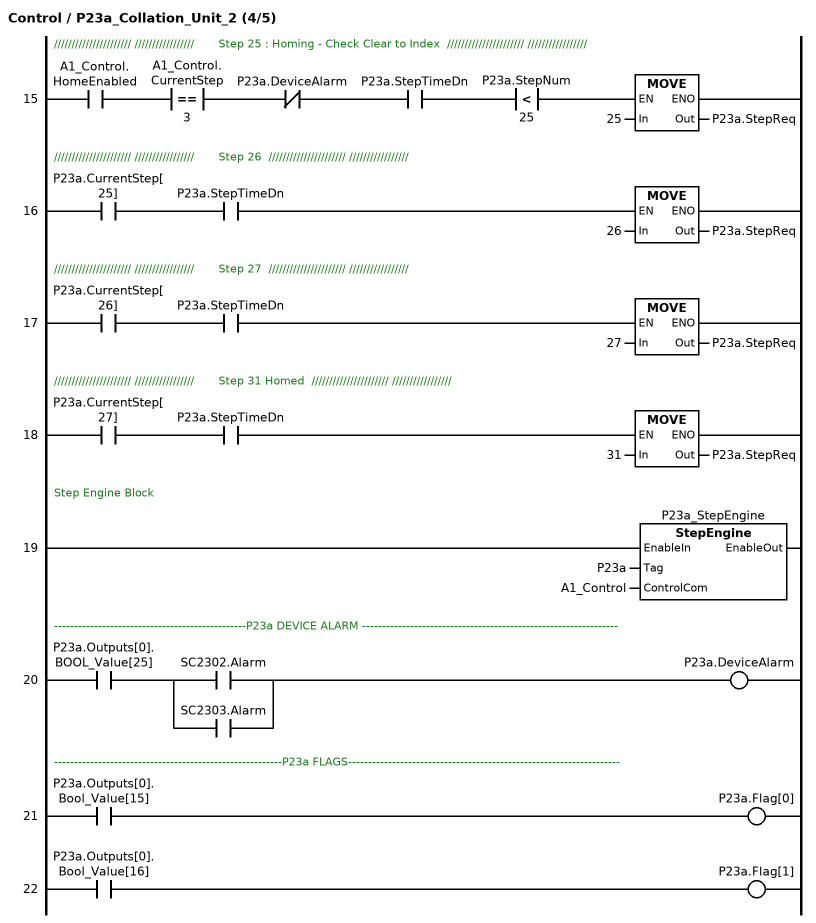
(* [picture p48: Control / P23a_Collation_Unit_2, rungs 15-22] *)
(* Rung 15: ////////////////////// /////////////////       Step 25 : Homing - Check Clear to Index  ////////////////////// ///////////////// *)
IF A1_Control.HomeEnabled AND (A1_Control.CurrentStep = 3) AND NOT P23a.DeviceAlarm AND P23a.StepTimeDn AND (P23a.StepNum < 25) THEN
    P23a.StepReq := 25;
END_IF;
(* Rung 16: ////////////////////// /////////////////       Step 26  ////////////////////// ///////////////// *)
IF P23a.CurrentStep[25] AND P23a.StepTimeDn THEN P23a.StepReq := 26; END_IF;
(* Rung 17: ////////////////////// /////////////////       Step 27  ////////////////////// ///////////////// *)
IF P23a.CurrentStep[26] AND P23a.StepTimeDn THEN P23a.StepReq := 27; END_IF;
(* Rung 18: ////////////////////// /////////////////       Step 31 Homed  ////////////////////// ///////////////// *)
IF P23a.CurrentStep[27] AND P23a.StepTimeDn THEN P23a.StepReq := 31; END_IF;
(* Rung 19: Step Engine Block *)
P23a_StepEngine(EnableIn := TRUE, Tag := P23a, ControlCom := A1_Control);
(* Rung 20: ------------------------------------------------P23a DEVICE ALARM ---------------------------------------------------------------- *)
P23a.DeviceAlarm := P23a.Outputs[0].BOOL_Value[25] AND (SC2302.Alarm OR SC2303.Alarm);
(* Rung 21: ---------------------------------------------------------P23a FLAGS-------------------------------------------------------------------- *)
P23a.Flag[0] := P23a.Outputs[0].Bool_Value[15];
(* Rung 22 *)
P23a.Flag[1] := P23a.Outputs[0].Bool_Value[16];

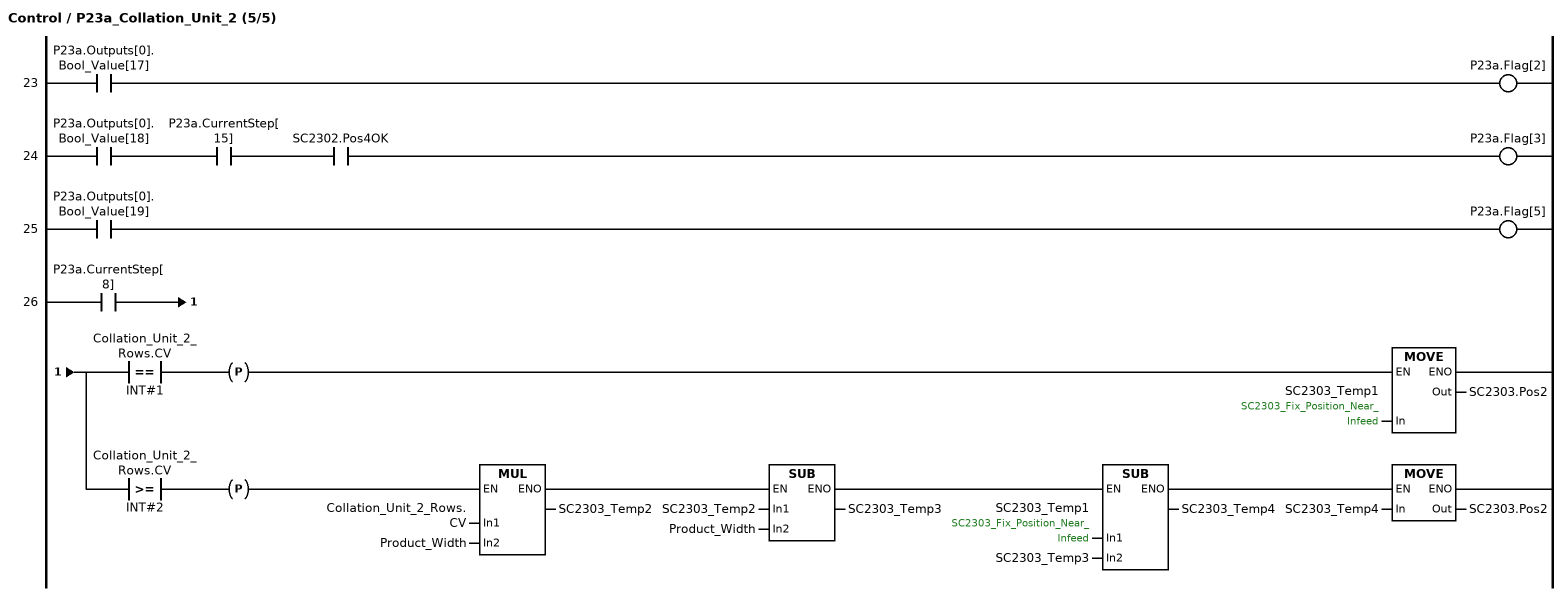
(* Rung 23 *)
P23a.Flag[2] := P23a.Outputs[0].Bool_Value[17];
(* Rung 24 *)
P23a.Flag[3] := P23a.Outputs[0].Bool_Value[18] AND P23a.CurrentStep[15] AND SC2302.Pos4OK;
(* notes on elements: Flag to Infeed conveyor *)
(* Rung 25 *)
P23a.Flag[5] := P23a.Outputs[0].Bool_Value[19];
(* Rung 26 *)
_e52(CLK := P23a.CurrentStep[8] AND (Collation_Unit_2_Rows.CV = INT#1));
IF _e52.Q THEN SC2303.Pos2 := SC2303_Temp1; END_IF;
_e53(CLK := P23a.CurrentStep[8] AND (Collation_Unit_2_Rows.CV >= INT#2));
IF _e53.Q THEN
    SC2303_Temp2 := Collation_Unit_2_Rows.CV * Product_Width;
    SC2303_Temp3 := SC2303_Temp2 - Product_Width;
    SC2303_Temp4 := SC2303_Temp1 - SC2303_Temp3;
    SC2303.Pos2 := SC2303_Temp4;
END_IF;

(* Section P17_MainDrive: ladder, written here as Structured Text *)

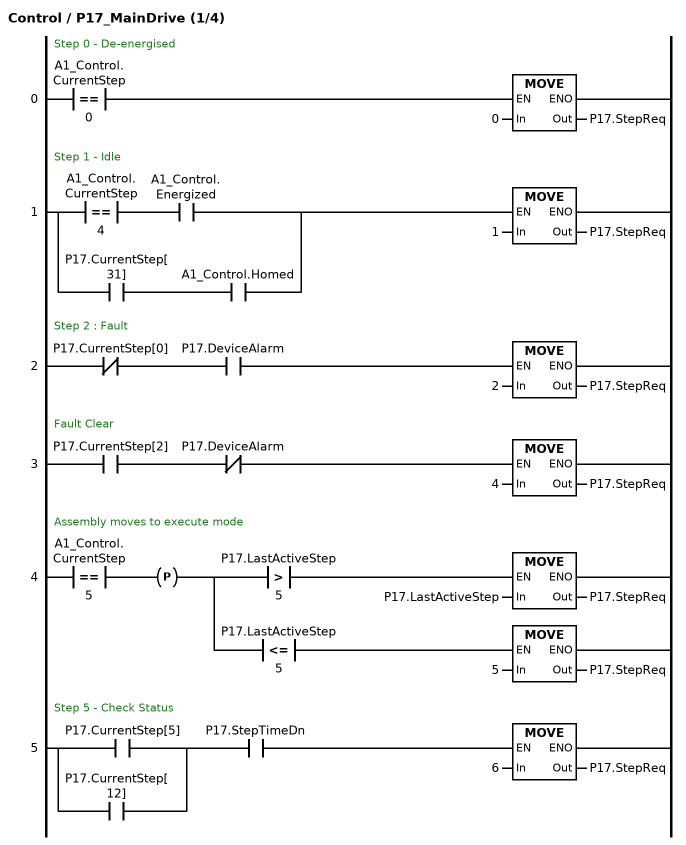
(* Rung 0: Step 0 - De-energised *)
IF A1_Control.CurrentStep = 0 THEN P17.StepReq := 0; END_IF;
(* Rung 1: Step 1 - Idle *)
IF ((A1_Control.CurrentStep = 4) AND A1_Control.Energized) OR (P17.CurrentStep[31] AND A1_Control.Homed) THEN
    P17.StepReq := 1;
END_IF;
(* Rung 2: Step 2 : Fault *)
IF NOT P17.CurrentStep[0] AND P17.DeviceAlarm THEN P17.StepReq := 2; END_IF;
(* Rung 3: Fault Clear *)
IF P17.CurrentStep[2] AND NOT P17.DeviceAlarm THEN P17.StepReq := 4; END_IF;
(* Rung 4: Assembly moves to execute mode *)
_e54(CLK := A1_Control.CurrentStep = 5);
IF _e54.Q AND (P17.LastActiveStep > 5) THEN P17.StepReq := P17.LastActiveStep; END_IF;
IF _e54.Q AND (P17.LastActiveStep <= 5) THEN P17.StepReq := 5; END_IF;
(* Rung 5: Step 5 - Check Status *)
IF (P17.CurrentStep[5] OR P17.CurrentStep[12]) AND P17.StepTimeDn THEN P17.StepReq := 6; END_IF;

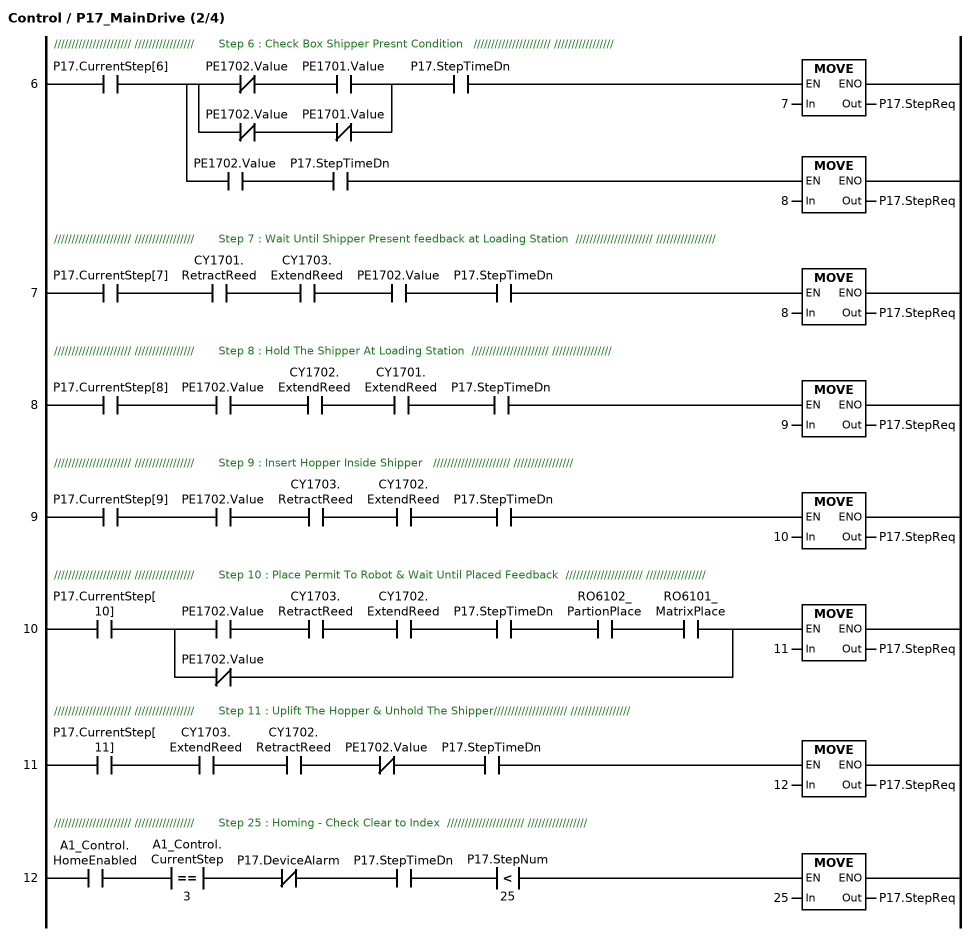
(* Rung 6: ////////////////////// /////////////////       Step 6 : Check Box Shipper Presnt Condition   ////////////////////// ///////////////// *)
_p55 := P17.CurrentStep[6];
IF P17.CurrentStep[6] AND ((NOT PE1702.Value AND PE1701.Value) OR (NOT PE1702.Value AND NOT PE1701.Value)) AND P17.StepTimeDn THEN
    P17.StepReq := 7;
END_IF;
IF _p55 AND PE1702.Value AND P17.StepTimeDn THEN P17.StepReq := 8; END_IF;
(* Rung 7: ////////////////////// /////////////////       Step 7 : Wait Until Shipper Present feedback at Loading Station  ////////////////////// ///////////////// *)
IF P17.CurrentStep[7] AND CY1701.RetractReed AND CY1703.ExtendReed AND PE1702.Value AND P17.StepTimeDn THEN
    P17.StepReq := 8;
END_IF;
(* Rung 8: ////////////////////// /////////////////       Step 8 : Hold The Shipper At Loading Station  ////////////////////// ///////////////// *)
IF P17.CurrentStep[8] AND PE1702.Value AND CY1702.ExtendReed AND CY1701.ExtendReed AND P17.StepTimeDn THEN
    P17.StepReq := 9;
END_IF;
(* Rung 9: ////////////////////// /////////////////       Step 9 : Insert Hopper Inside Shipper   ////////////////////// ///////////////// *)
IF P17.CurrentStep[9] AND PE1702.Value AND CY1703.RetractReed AND CY1702.ExtendReed AND P17.StepTimeDn THEN
    P17.StepReq := 10;
END_IF;
(* Rung 10: ////////////////////// /////////////////       Step 10 : Place Permit To Robot & Wait Until Placed Feedback  ////////////////////// ///////////////// *)
IF P17.CurrentStep[10] AND ((PE1702.Value AND CY1703.RetractReed AND CY1702.ExtendReed AND P17.StepTimeDn AND RO6102_PartionPlace AND RO6101_MatrixPlace) OR NOT PE1702.Value) THEN
    P17.StepReq := 11;
END_IF;
(* Rung 11: ////////////////////// /////////////////       Step 11 : Uplift The Hopper & Unhold The Shipper///////////////////// ///////////////// *)
IF P17.CurrentStep[11] AND CY1703.ExtendReed AND CY1702.RetractReed AND NOT PE1702.Value AND P17.StepTimeDn THEN
    P17.StepReq := 12;
END_IF;
(* Rung 12: ////////////////////// /////////////////       Step 25 : Homing - Check Clear to Index  ////////////////////// ///////////////// *)
IF A1_Control.HomeEnabled AND (A1_Control.CurrentStep = 3) AND NOT P17.DeviceAlarm AND P17.StepTimeDn AND (P17.StepNum < 25) THEN
    P17.StepReq := 25;
END_IF;

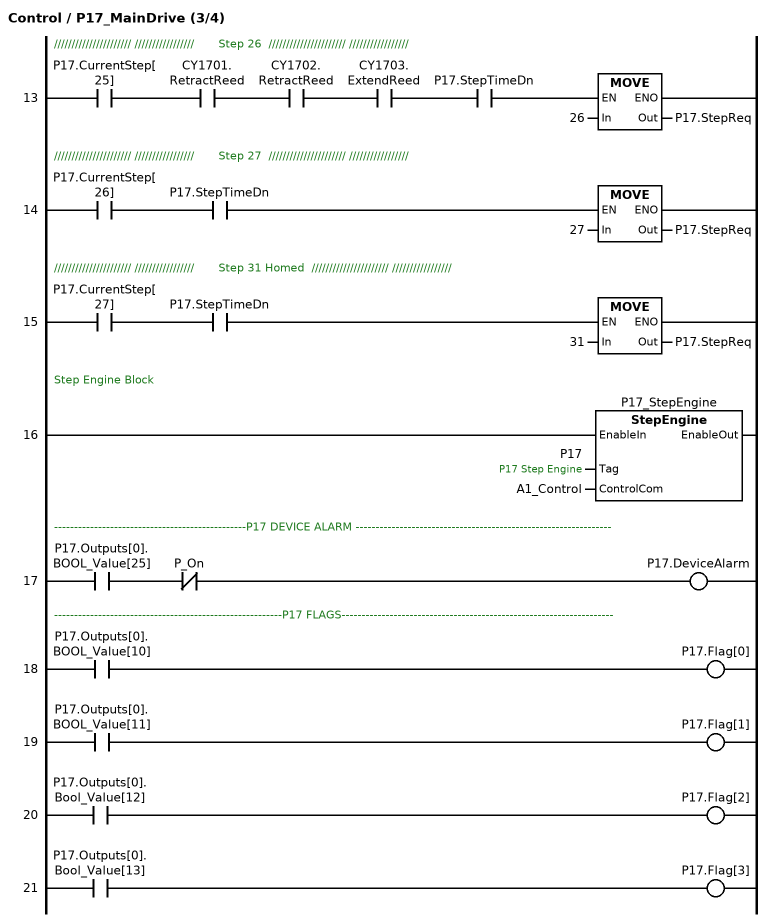
(* Rung 13: ////////////////////// /////////////////       Step 26  ////////////////////// ///////////////// *)
IF P17.CurrentStep[25] AND CY1701.RetractReed AND CY1702.RetractReed AND CY1703.ExtendReed AND P17.StepTimeDn THEN
    P17.StepReq := 26;
END_IF;
(* Rung 14: ////////////////////// /////////////////       Step 27  ////////////////////// ///////////////// *)
IF P17.CurrentStep[26] AND P17.StepTimeDn THEN P17.StepReq := 27; END_IF;
(* Rung 15: ////////////////////// /////////////////       Step 31 Homed  ////////////////////// ///////////////// *)
IF P17.CurrentStep[27] AND P17.StepTimeDn THEN P17.StepReq := 31; END_IF;
(* Rung 16: Step Engine Block *)
P17_StepEngine(EnableIn := TRUE, Tag := P17, ControlCom := A1_Control);
(* Rung 17: ------------------------------------------------P17 DEVICE ALARM ---------------------------------------------------------------- *)
P17.DeviceAlarm := P17.Outputs[0].BOOL_Value[25] AND NOT P_On;
(* Rung 18: ---------------------------------------------------------P17 FLAGS-------------------------------------------------------------------- *)
P17.Flag[0] := P17.Outputs[0].BOOL_Value[10];
(* Rung 19 *)
P17.Flag[1] := P17.Outputs[0].BOOL_Value[11];
(* Rung 20 *)
P17.Flag[2] := P17.Outputs[0].Bool_Value[12];
(* Rung 21 *)
P17.Flag[3] := P17.Outputs[0].Bool_Value[13];

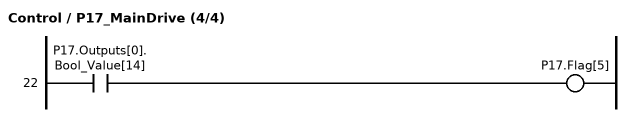
(* Rung 22 *)
P17.Flag[5] := P17.Outputs[0].Bool_Value[14];

(* Section P27_TopTapping: ladder, written here as Structured Text *)

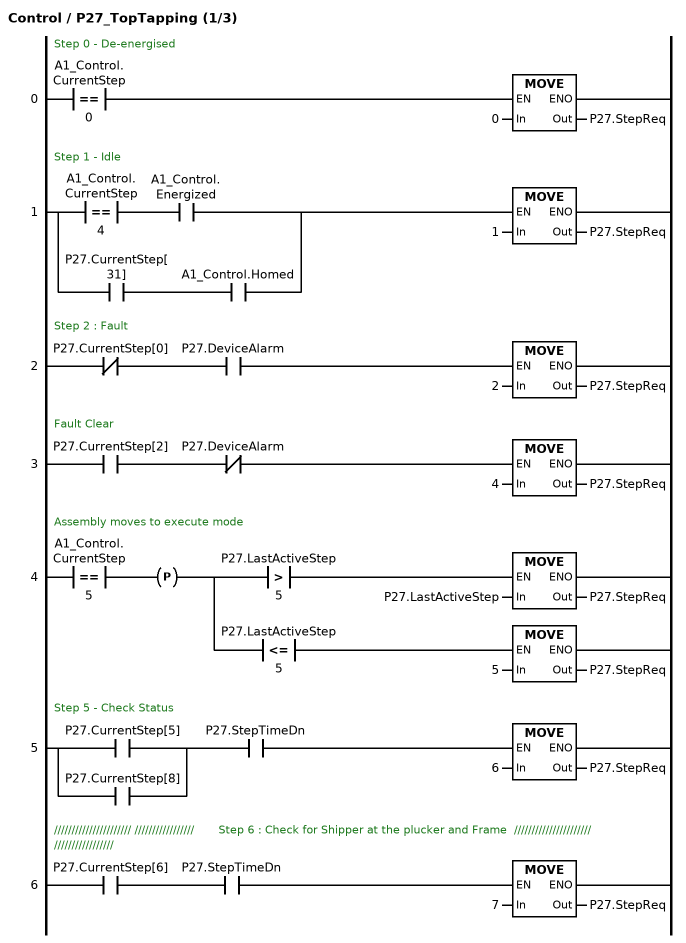
(* Rung 0: Step 0 - De-energised *)
IF A1_Control.CurrentStep = 0 THEN P27.StepReq := 0; END_IF;
(* Rung 1: Step 1 - Idle *)
IF ((A1_Control.CurrentStep = 4) AND A1_Control.Energized) OR (P27.CurrentStep[31] AND A1_Control.Homed) THEN
    P27.StepReq := 1;
END_IF;
(* Rung 2: Step 2 : Fault *)
IF NOT P27.CurrentStep[0] AND P27.DeviceAlarm THEN P27.StepReq := 2; END_IF;
(* Rung 3: Fault Clear *)
IF P27.CurrentStep[2] AND NOT P27.DeviceAlarm THEN P27.StepReq := 4; END_IF;
(* Rung 4: Assembly moves to execute mode *)
_e56(CLK := A1_Control.CurrentStep = 5);
IF _e56.Q AND (P27.LastActiveStep > 5) THEN P27.StepReq := P27.LastActiveStep; END_IF;
IF _e56.Q AND (P27.LastActiveStep <= 5) THEN P27.StepReq := 5; END_IF;
(* Rung 5: Step 5 - Check Status *)
IF (P27.CurrentStep[5] OR P27.CurrentStep[8]) AND P27.StepTimeDn THEN P27.StepReq := 6; END_IF;
(* Rung 6: ////////////////////// /////////////////       Step 6 : Check for Shipper at the plucker and Frame  ////////////////////// ///////////////// *)
IF P27.CurrentStep[6] AND P27.StepTimeDn THEN P27.StepReq := 7; END_IF;

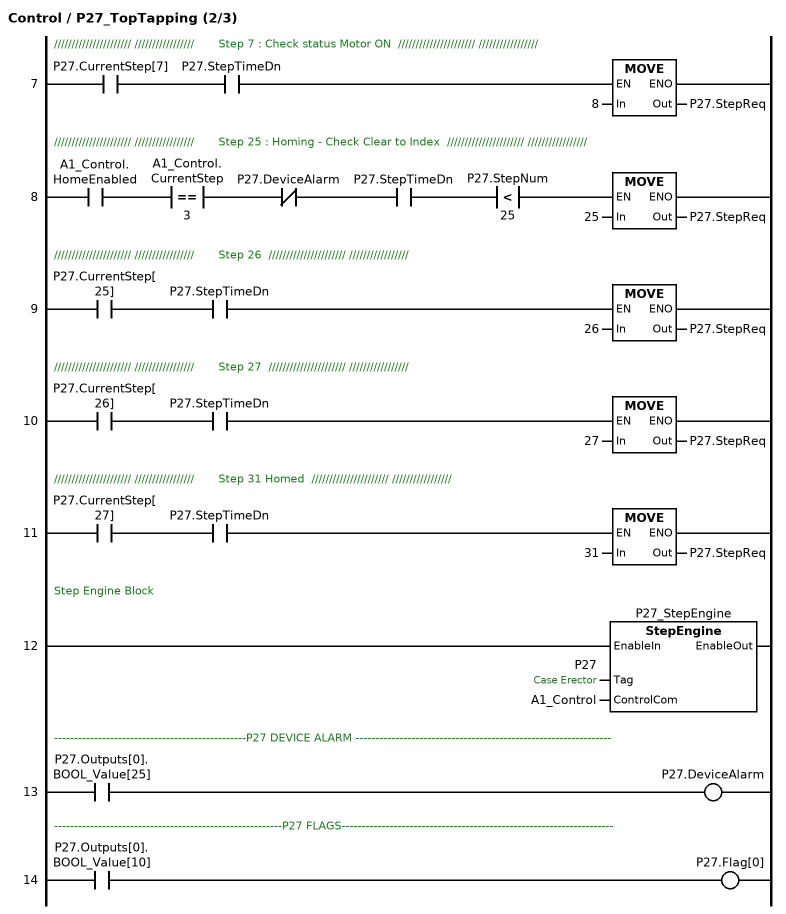
(* Rung 7: ////////////////////// /////////////////       Step 7 : Check status Motor ON  ////////////////////// ///////////////// *)
IF P27.CurrentStep[7] AND P27.StepTimeDn THEN P27.StepReq := 8; END_IF;
(* Rung 8: ////////////////////// /////////////////       Step 25 : Homing - Check Clear to Index  ////////////////////// ///////////////// *)
IF A1_Control.HomeEnabled AND (A1_Control.CurrentStep = 3) AND NOT P27.DeviceAlarm AND P27.StepTimeDn AND (P27.StepNum < 25) THEN
    P27.StepReq := 25;
END_IF;
(* Rung 9: ////////////////////// /////////////////       Step 26  ////////////////////// ///////////////// *)
IF P27.CurrentStep[25] AND P27.StepTimeDn THEN P27.StepReq := 26; END_IF;
(* Rung 10: ////////////////////// /////////////////       Step 27  ////////////////////// ///////////////// *)
IF P27.CurrentStep[26] AND P27.StepTimeDn THEN P27.StepReq := 27; END_IF;
(* Rung 11: ////////////////////// /////////////////       Step 31 Homed  ////////////////////// ///////////////// *)
IF P27.CurrentStep[27] AND P27.StepTimeDn THEN P27.StepReq := 31; END_IF;
(* Rung 12: Step Engine Block *)
P27_StepEngine(EnableIn := TRUE, Tag := P27, ControlCom := A1_Control);
(* Rung 13: ------------------------------------------------P27 DEVICE ALARM ---------------------------------------------------------------- *)
P27.DeviceAlarm := P27.Outputs[0].BOOL_Value[25];
(* Rung 14: ---------------------------------------------------------P27 FLAGS-------------------------------------------------------------------- *)
P27.Flag[0] := P27.Outputs[0].BOOL_Value[10];

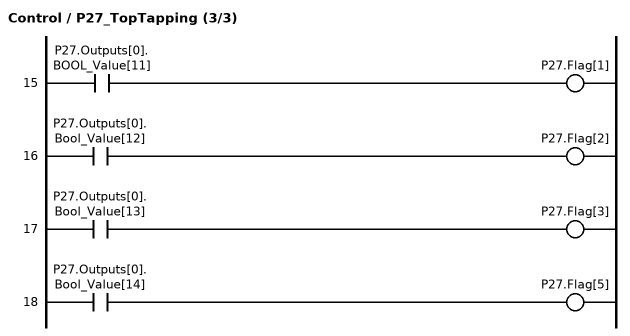
(* Rung 15 *)
P27.Flag[1] := P27.Outputs[0].BOOL_Value[11];
(* Rung 16 *)
P27.Flag[2] := P27.Outputs[0].Bool_Value[12];
(* Rung 17 *)
P27.Flag[3] := P27.Outputs[0].Bool_Value[13];
(* Rung 18 *)
P27.Flag[5] := P27.Outputs[0].Bool_Value[14];

(* Section P71_RotaryRoller: ladder, written here as Structured Text *)

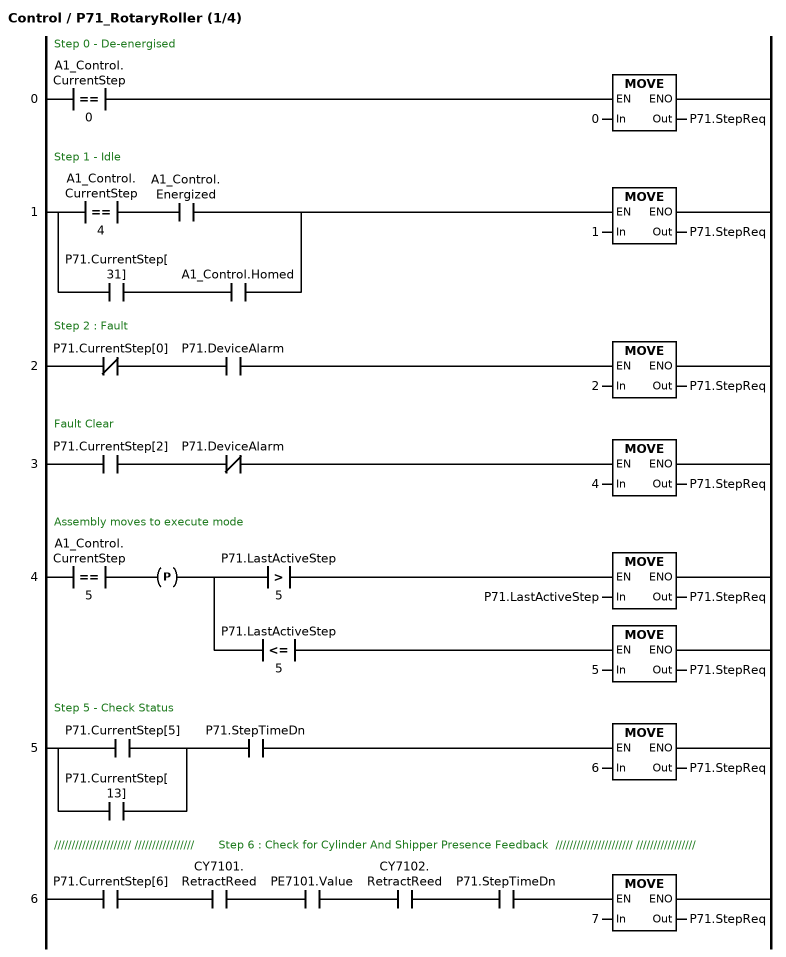
(* Rung 0: Step 0 - De-energised *)
IF A1_Control.CurrentStep = 0 THEN P71.StepReq := 0; END_IF;
(* Rung 1: Step 1 - Idle *)
IF ((A1_Control.CurrentStep = 4) AND A1_Control.Energized) OR (P71.CurrentStep[31] AND A1_Control.Homed) THEN
    P71.StepReq := 1;
END_IF;
(* Rung 2: Step 2 : Fault *)
IF NOT P71.CurrentStep[0] AND P71.DeviceAlarm THEN P71.StepReq := 2; END_IF;
(* Rung 3: Fault Clear *)
IF P71.CurrentStep[2] AND NOT P71.DeviceAlarm THEN P71.StepReq := 4; END_IF;
(* Rung 4: Assembly moves to execute mode *)
_e57(CLK := A1_Control.CurrentStep = 5);
IF _e57.Q AND (P71.LastActiveStep > 5) THEN P71.StepReq := P71.LastActiveStep; END_IF;
IF _e57.Q AND (P71.LastActiveStep <= 5) THEN P71.StepReq := 5; END_IF;
(* Rung 5: Step 5 - Check Status *)
IF (P71.CurrentStep[5] OR P71.CurrentStep[13]) AND P71.StepTimeDn THEN P71.StepReq := 6; END_IF;
(* Rung 6: ////////////////////// /////////////////       Step 6 : Check for Cylinder And Shipper Presence Feedback  ////////////////////// ///////////////// *)
IF P71.CurrentStep[6] AND CY7101.RetractReed AND PE7101.Value AND CY7102.RetractReed AND P71.StepTimeDn THEN
    P71.StepReq := 7;
END_IF;

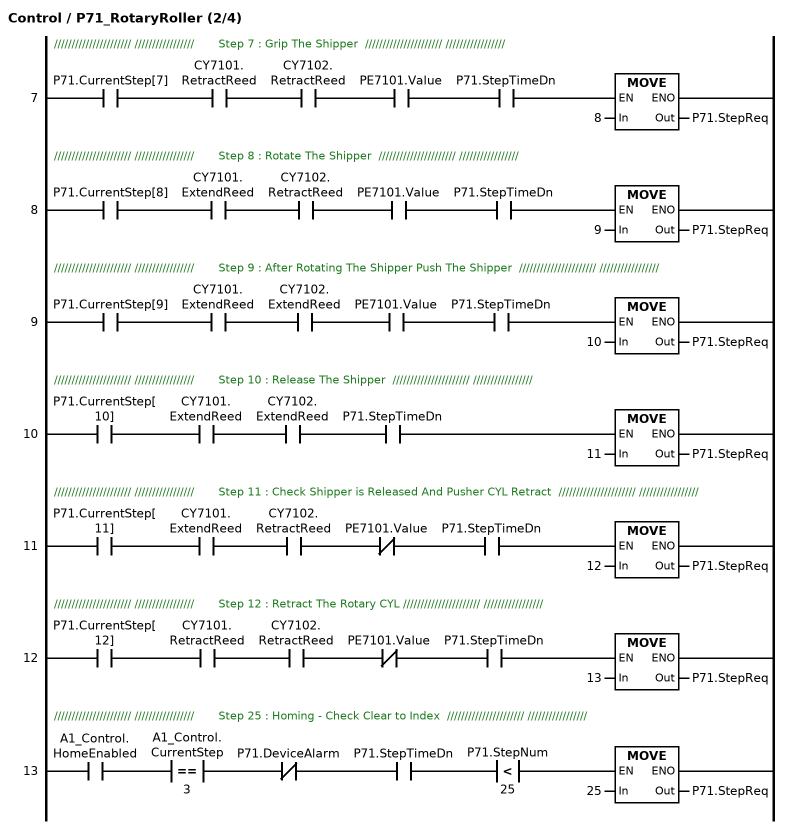
(* Rung 7: ////////////////////// /////////////////       Step 7 : Grip The Shipper  ////////////////////// ///////////////// *)
IF P71.CurrentStep[7] AND CY7101.RetractReed AND CY7102.RetractReed AND PE7101.Value AND P71.StepTimeDn THEN
    P71.StepReq := 8;
END_IF;
(* Rung 8: ////////////////////// /////////////////       Step 8 : Rotate The Shipper  ////////////////////// ///////////////// *)
IF P71.CurrentStep[8] AND CY7101.ExtendReed AND CY7102.RetractReed AND PE7101.Value AND P71.StepTimeDn THEN
    P71.StepReq := 9;
END_IF;
(* Rung 9: ////////////////////// /////////////////       Step 9 : After Rotating The Shipper Push The Shipper  ////////////////////// ///////////////// *)
IF P71.CurrentStep[9] AND CY7101.ExtendReed AND CY7102.ExtendReed AND PE7101.Value AND P71.StepTimeDn THEN
    P71.StepReq := 10;
END_IF;
(* Rung 10: ////////////////////// /////////////////       Step 10 : Release The Shipper  ////////////////////// ///////////////// *)
IF P71.CurrentStep[10] AND CY7101.ExtendReed AND CY7102.ExtendReed AND P71.StepTimeDn THEN
    P71.StepReq := 11;
END_IF;
(* Rung 11: ////////////////////// /////////////////       Step 11 : Check Shipper is Released And Pusher CYL Retract  ////////////////////// ///////////////// *)
IF P71.CurrentStep[11] AND CY7101.ExtendReed AND CY7102.RetractReed AND NOT PE7101.Value AND P71.StepTimeDn THEN
    P71.StepReq := 12;
END_IF;
(* Rung 12: ////////////////////// /////////////////       Step 12 : Retract The Rotary CYL ////////////////////// ///////////////// *)
IF P71.CurrentStep[12] AND CY7101.RetractReed AND CY7102.RetractReed AND NOT PE7101.Value AND P71.StepTimeDn THEN
    P71.StepReq := 13;
END_IF;
(* Rung 13: ////////////////////// /////////////////       Step 25 : Homing - Check Clear to Index  ////////////////////// ///////////////// *)
IF A1_Control.HomeEnabled AND (A1_Control.CurrentStep = 3) AND NOT P71.DeviceAlarm AND P71.StepTimeDn AND (P71.StepNum < 25) THEN
    P71.StepReq := 25;
END_IF;

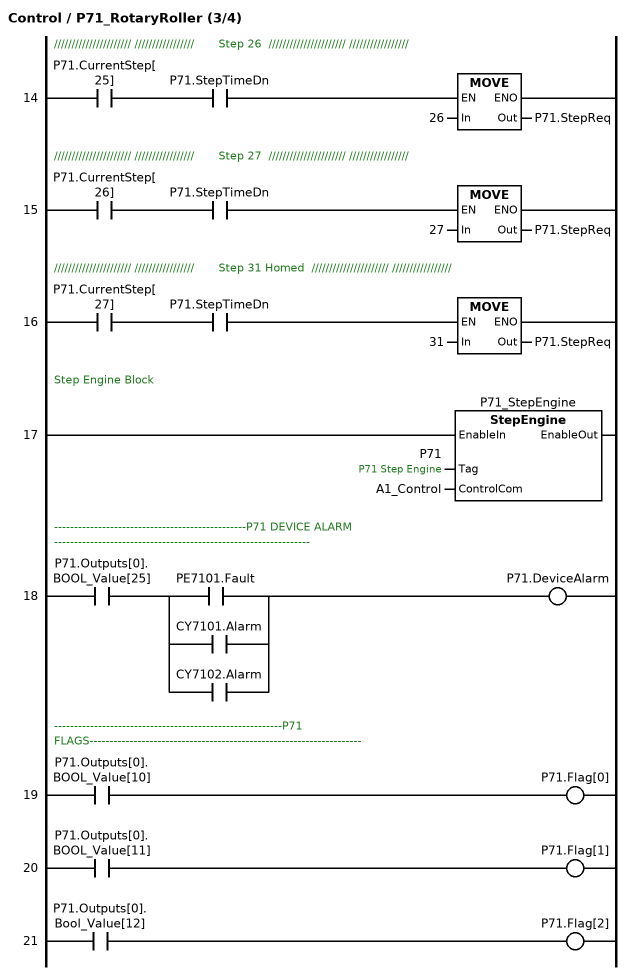
(* Rung 14: ////////////////////// /////////////////       Step 26  ////////////////////// ///////////////// *)
IF P71.CurrentStep[25] AND P71.StepTimeDn THEN P71.StepReq := 26; END_IF;
(* Rung 15: ////////////////////// /////////////////       Step 27  ////////////////////// ///////////////// *)
IF P71.CurrentStep[26] AND P71.StepTimeDn THEN P71.StepReq := 27; END_IF;
(* Rung 16: ////////////////////// /////////////////       Step 31 Homed  ////////////////////// ///////////////// *)
IF P71.CurrentStep[27] AND P71.StepTimeDn THEN P71.StepReq := 31; END_IF;
(* Rung 17: Step Engine Block *)
P71_StepEngine(EnableIn := TRUE, Tag := P71, ControlCom := A1_Control);
(* Rung 18: ------------------------------------------------P71 DEVICE ALARM ---------------------------------------------------------------- *)
P71.DeviceAlarm := P71.Outputs[0].BOOL_Value[25] AND (PE7101.Fault OR CY7101.Alarm OR CY7102.Alarm);
(* Rung 19: ---------------------------------------------------------P71 FLAGS-------------------------------------------------------------------- *)
P71.Flag[0] := P71.Outputs[0].BOOL_Value[10];
(* Rung 20 *)
P71.Flag[1] := P71.Outputs[0].BOOL_Value[11];
(* Rung 21 *)
P71.Flag[2] := P71.Outputs[0].Bool_Value[12];

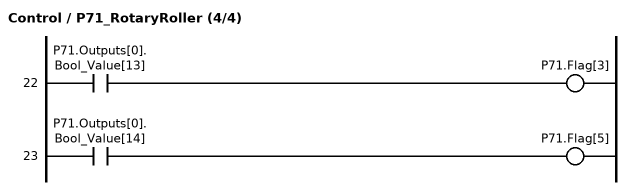
(* Rung 22 *)
P71.Flag[3] := P71.Outputs[0].Bool_Value[13];
(* Rung 23 *)
P71.Flag[5] := P71.Outputs[0].Bool_Value[14];

(* Section P34_Label_Conveyor: ladder, written here as Structured Text *)

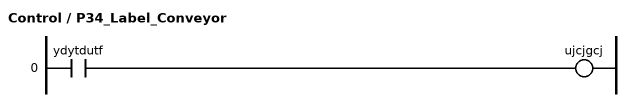
(* Rung 0 *)
ujcjgcj := ydytdutf;

(* Section RO6301: ladder, written here as Structured Text *)

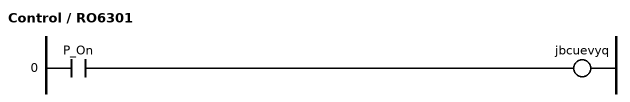
(* Rung 0 *)
jbcuevyq := P_On;

(* Section RO6302: ladder, written here as Structured Text *)

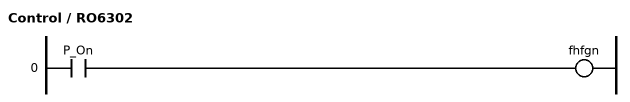
(* Rung 0 *)
fhfgn := P_On;

(* Section RO6303: ladder, written here as Structured Text *)

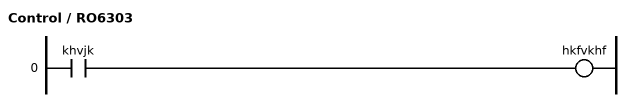
(* Rung 0 *)
hkfvkhf := khvjk;

(* Section Statistics: ladder, written here as Structured Text *)

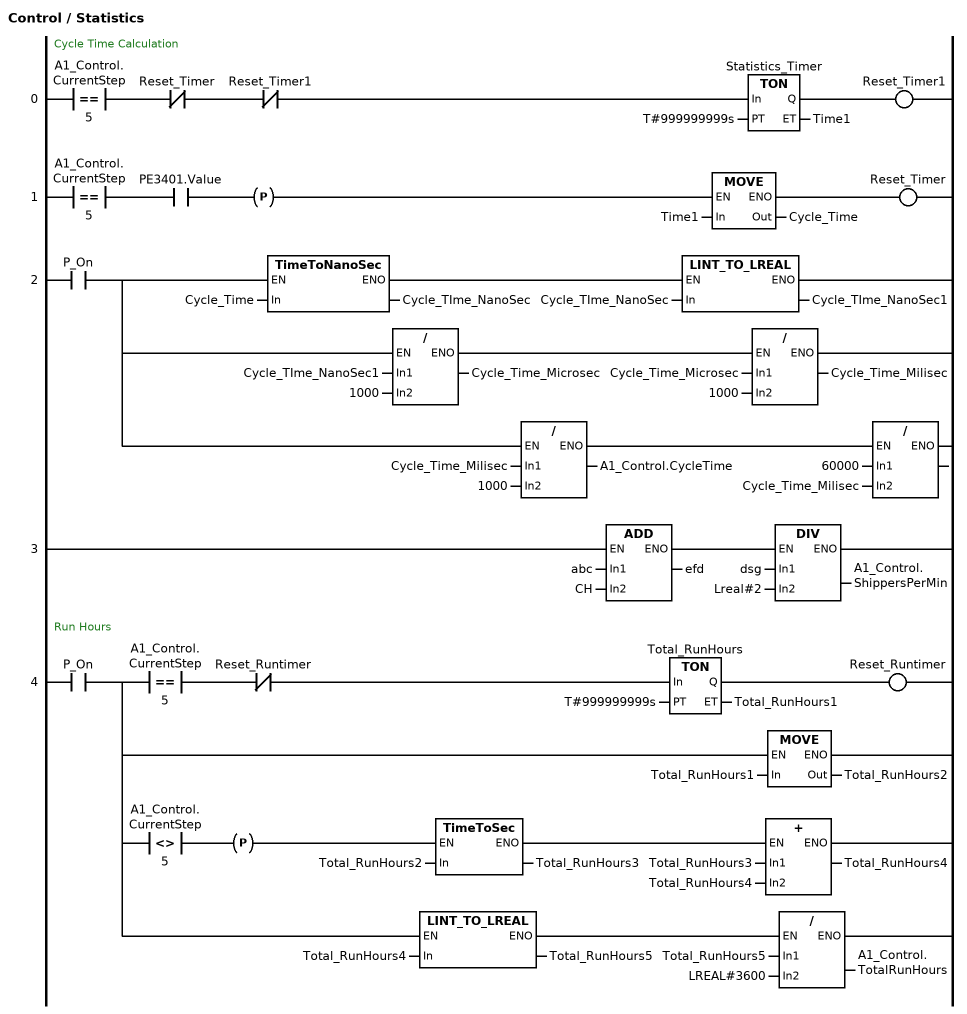
(* Rung 0: Cycle Time Calculation *)
Statistics_Timer(In := (A1_Control.CurrentStep = 5) AND NOT Reset_Timer AND NOT Reset_Timer1, PT := T#999999999s, ET => Time1);
Reset_Timer1 := Statistics_Timer.Q;
(* Rung 1 *)
_e58(CLK := (A1_Control.CurrentStep = 5) AND PE3401.Value);
IF _e58.Q THEN Cycle_Time := Time1; END_IF;
Reset_Timer := _e58.Q;
(* Rung 2 *)
IF P_On THEN
    Cycle_TIme_NanoSec := TimeToNanoSec(In := Cycle_Time);
    Cycle_TIme_NanoSec1 := LINT_TO_LREAL(In := Cycle_TIme_NanoSec);
    Cycle_Time_Microsec := Cycle_TIme_NanoSec1 / 1000;
    Cycle_Time_Milisec := Cycle_Time_Microsec / 1000;
    A1_Control.CycleTime := Cycle_Time_Milisec / 1000;
    _t59 := 60000 / Cycle_Time_Milisec;
END_IF;
(* Rung 3 *)
efd := abc + CH;
A1_Control.ShippersPerMin := dsg / Lreal#2;
(* Rung 4: Run Hours *)
Total_RunHours(In := P_On AND (A1_Control.CurrentStep = 5) AND NOT Reset_Runtimer, PT := T#999999999s, ET => Total_RunHours1);
Reset_Runtimer := Total_RunHours.Q;
IF P_On THEN Total_RunHours2 := Total_RunHours1; END_IF;
_e60(CLK := P_On AND (A1_Control.CurrentStep <> 5));
IF _e60.Q THEN
    Total_RunHours3 := TimeToSec(In := Total_RunHours2);
    Total_RunHours4 := Total_RunHours3 + Total_RunHours4;
END_IF;
IF P_On THEN
    Total_RunHours5 := LINT_TO_LREAL(In := Total_RunHours4);
    A1_Control.TotalRunHours := Total_RunHours5 / LREAL#3600;
END_IF;

(* Section Recipes: ladder, written here as Structured Text *)

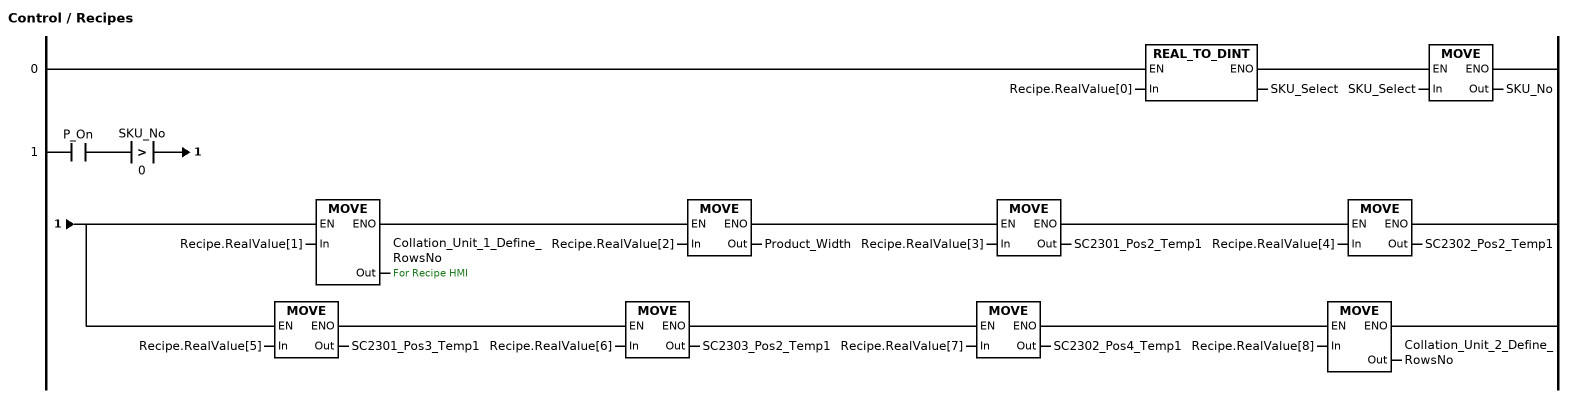
(* Rung 0 *)
SKU_Select := REAL_TO_DINT(In := Recipe.RealValue[0]);
SKU_No := SKU_Select;
(* Rung 1 *)
IF P_On AND (SKU_No > 0) THEN
    Collation_Unit_1_Define_RowsNo := Recipe.RealValue[1];
    Product_Width := Recipe.RealValue[2];
    SC2301_Pos2_Temp1 := Recipe.RealValue[3];
    SC2302_Pos2_Temp1 := Recipe.RealValue[4];
    SC2301_Pos3_Temp1 := Recipe.RealValue[5];
    SC2303_Pos2_Temp1 := Recipe.RealValue[6];
    SC2302_Pos4_Temp1 := Recipe.RealValue[7];
    Collation_Unit_2_Define_RowsNo := Recipe.RealValue[8];
END_IF;

(* Section BatchReporting: ladder, written here as Structured Text *)

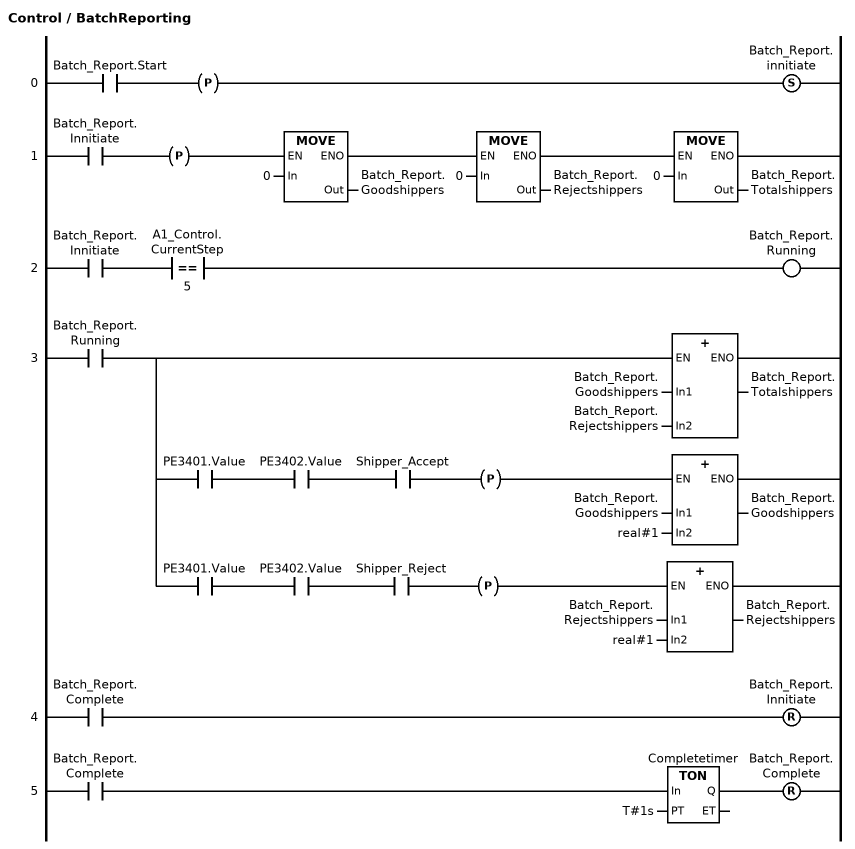
(* Rung 0 *)
_e61(CLK := Batch_Report.Start);
IF _e61.Q THEN Batch_Report.innitiate := TRUE; END_IF;
(* Rung 1 *)
_e62(CLK := Batch_Report.Innitiate);
IF _e62.Q THEN
    Batch_Report.Goodshippers := 0;
    Batch_Report.Rejectshippers := 0;
    Batch_Report.Totalshippers := 0;
END_IF;
(* Rung 2 *)
Batch_Report.Running := Batch_Report.Innitiate AND (A1_Control.CurrentStep = 5);
(* Rung 3 *)
_p63 := Batch_Report.Running;
IF _p63 THEN
    Batch_Report.Totalshippers := Batch_Report.Goodshippers + Batch_Report.Rejectshippers;
END_IF;
_e64(CLK := _p63 AND PE3401.Value AND PE3402.Value AND Shipper_Accept);
IF _e64.Q THEN Batch_Report.Goodshippers := Batch_Report.Goodshippers + real#1; END_IF;
_e65(CLK := _p63 AND PE3401.Value AND PE3402.Value AND Shipper_Reject);
IF _e65.Q THEN Batch_Report.Rejectshippers := Batch_Report.Rejectshippers + real#1; END_IF;
(* Rung 4 *)
IF Batch_Report.Complete THEN Batch_Report.Innitiate := FALSE; END_IF;
(* Rung 5 *)
Completetimer(In := Batch_Report.Complete, PT := T#1s);
IF Completetimer.Q THEN Batch_Report.Complete := FALSE; END_IF;

(* Section SequenceCylinder: ladder, written here as Structured Text *)

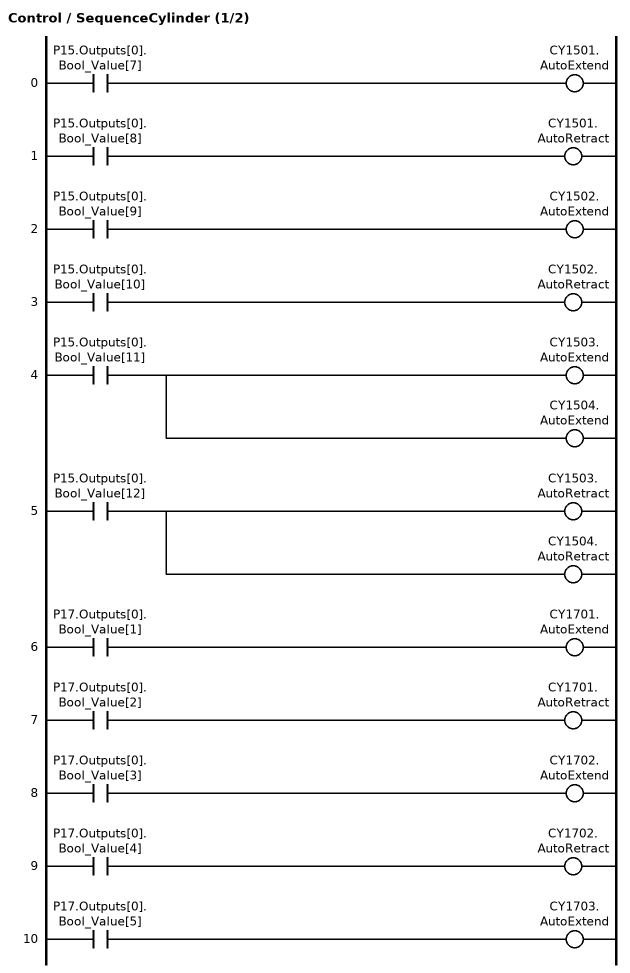
(* Rung 0 *)
CY1501.AutoExtend := P15.Outputs[0].Bool_Value[7];
(* Rung 1 *)
CY1501.AutoRetract := P15.Outputs[0].Bool_Value[8];
(* Rung 2 *)
CY1502.AutoExtend := P15.Outputs[0].Bool_Value[9];
(* Rung 3 *)
CY1502.AutoRetract := P15.Outputs[0].Bool_Value[10];
(* Rung 4 *)
CY1503.AutoExtend := P15.Outputs[0].Bool_Value[11];
CY1504.AutoExtend := P15.Outputs[0].Bool_Value[11];
(* Rung 5 *)
CY1503.AutoRetract := P15.Outputs[0].Bool_Value[12];
CY1504.AutoRetract := P15.Outputs[0].Bool_Value[12];
(* Rung 6 *)
CY1701.AutoExtend := P17.Outputs[0].Bool_Value[1];
(* Rung 7 *)
CY1701.AutoRetract := P17.Outputs[0].Bool_Value[2];
(* Rung 8 *)
CY1702.AutoExtend := P17.Outputs[0].Bool_Value[3];
(* Rung 9 *)
CY1702.AutoRetract := P17.Outputs[0].Bool_Value[4];
(* Rung 10 *)
CY1703.AutoExtend := P17.Outputs[0].Bool_Value[5];

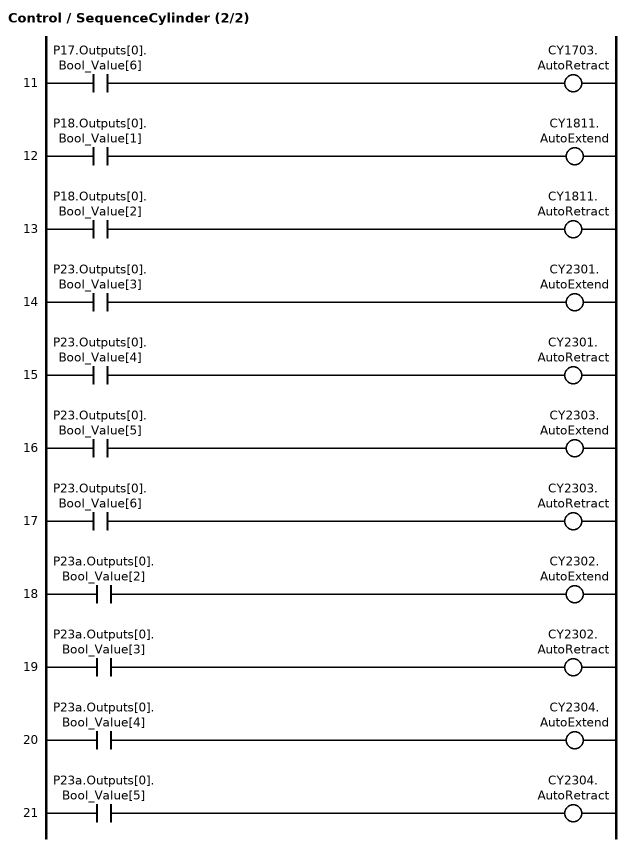
(* Rung 11 *)
CY1703.AutoRetract := P17.Outputs[0].Bool_Value[6];
(* Rung 12 *)
CY1811.AutoExtend := P18.Outputs[0].Bool_Value[1];
(* Rung 13 *)
CY1811.AutoRetract := P18.Outputs[0].Bool_Value[2];
(* Rung 14 *)
CY2301.AutoExtend := P23.Outputs[0].Bool_Value[3];
(* Rung 15 *)
CY2301.AutoRetract := P23.Outputs[0].Bool_Value[4];
(* Rung 16 *)
CY2303.AutoExtend := P23.Outputs[0].Bool_Value[5];
(* Rung 17 *)
CY2303.AutoRetract := P23.Outputs[0].Bool_Value[6];
(* Rung 18 *)
CY2302.AutoExtend := P23a.Outputs[0].Bool_Value[2];
(* Rung 19 *)
CY2302.AutoRetract := P23a.Outputs[0].Bool_Value[3];
(* Rung 20 *)
CY2304.AutoExtend := P23a.Outputs[0].Bool_Value[4];
(* Rung 21 *)
CY2304.AutoRetract := P23a.Outputs[0].Bool_Value[5];

(* Section SequenceMiscOut: ladder, written here as Structured Text *)

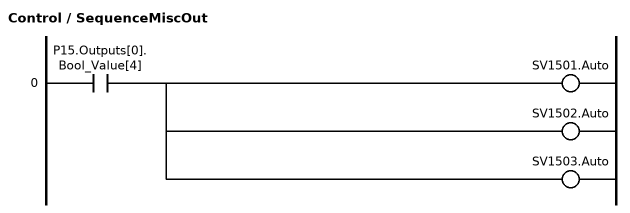
(* Rung 0 *)
SV1501.Auto := P15.Outputs[0].Bool_Value[4];
SV1502.Auto := P15.Outputs[0].Bool_Value[4];
SV1503.Auto := P15.Outputs[0].Bool_Value[4];

(* Section SequenceServo: ladder, written here as Structured Text *)

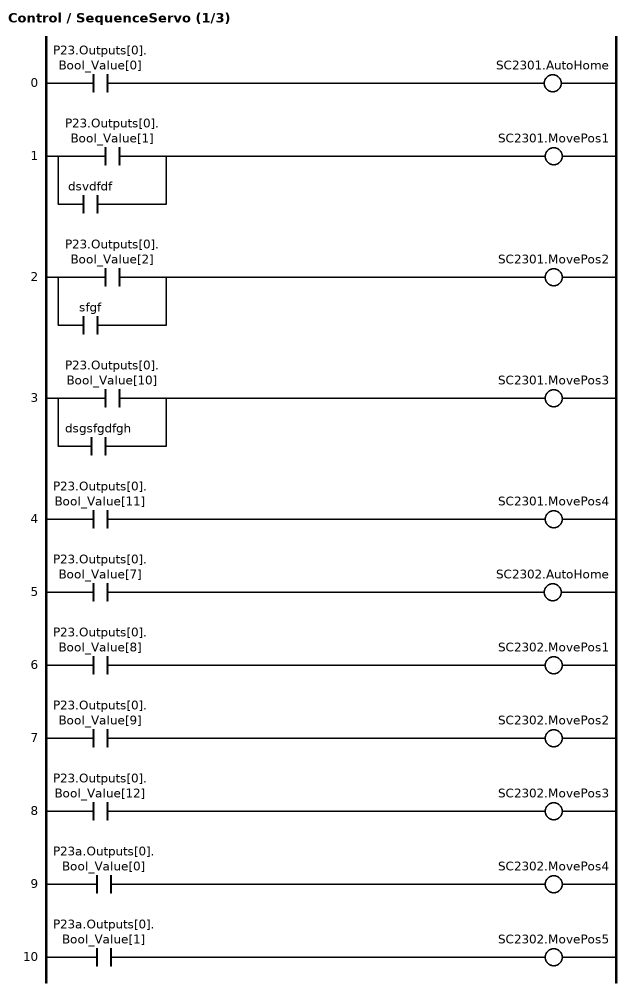
(* Rung 0 *)
SC2301.AutoHome := P23.Outputs[0].Bool_Value[0];
(* Rung 1 *)
SC2301.MovePos1 := P23.Outputs[0].Bool_Value[1] OR dsvdfdf;
(* Rung 2 *)
SC2301.MovePos2 := P23.Outputs[0].Bool_Value[2] OR sfgf;
(* Rung 3 *)
SC2301.MovePos3 := P23.Outputs[0].Bool_Value[10] OR dsgsfgdfgh;
(* Rung 4 *)
SC2301.MovePos4 := P23.Outputs[0].Bool_Value[11];
(* Rung 5 *)
SC2302.AutoHome := P23.Outputs[0].Bool_Value[7];
(* Rung 6 *)
SC2302.MovePos1 := P23.Outputs[0].Bool_Value[8];
(* Rung 7 *)
SC2302.MovePos2 := P23.Outputs[0].Bool_Value[9];
(* Rung 8 *)
SC2302.MovePos3 := P23.Outputs[0].Bool_Value[12];
(* Rung 9 *)
SC2302.MovePos4 := P23a.Outputs[0].Bool_Value[0];
(* Rung 10 *)
SC2302.MovePos5 := P23a.Outputs[0].Bool_Value[1];

